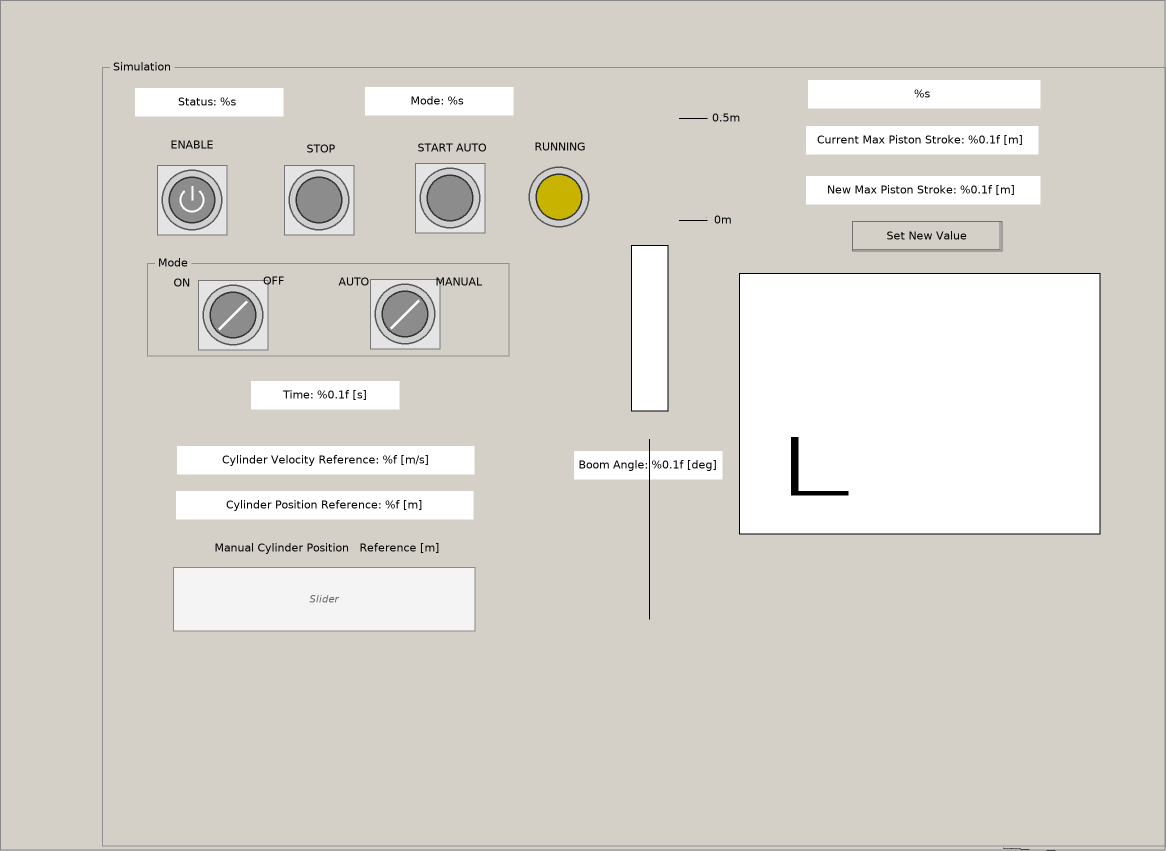
VISUALIZATION CraneHMI  // 1166x851
    Rectangle (566,310 166x37), angle 270
    GroupBox (102,59 1064x787), "Simulation"
        GroupBox (45,196 362x101), "Mode"
        Rectangle (637,214 361x261)
        PowerSwitch (55,106 70x70), variable: HMI.bPowerOn, behaviour: TOGGLE, style: Switch-PowerSwitch-Gray
        PushSwitch (313,104 70x70), variable: HMI.bStart, behaviour: TAP, style: Switch-PushSwitch-Gray
        Lamp1 (422,103 70x70), variable: HMI.bRunning, style: Lamp-Lamp1-Yellow
        Textfield (74,386 299x30), "Cylinder Velocity Reference: %f [m/s]", text variable: HMI.fCylinderVelocityReference
            OnMouseClick: write the text variable via Default
        Label (15,71 150x30), "ENABLE"
        Label (275,74 150x30), "START AUTO"
        Label (383,73 150x30), "RUNNING"
        Textfield (148,321 150x30), "Time: %0.1f [s]", text variable: HMI.fSimulationTime
        Label (90,474 270x30), "Manual Cylinder Position Reference [m]"
        Textfield (73,431 299x30), "Cylinder Position Reference: %f [m]", text variable: HMI.fCylinderPosition
        Line (577,161) (605,161)
        Label (607,146 28x30), "0m"
        Textfield (703,66 234x30), "Current Max Piston Stroke: %0.1f [m]", text variable: Parameters.stParam.stPistonRange.fPistonPosMax
        Textfield (703,116 236x30), "New Max Piston Stroke: %0.1f [m]", text variable: HMI.fMaxPistonPosition
            OnMouseDown: write the text variable via Default, min 0, max 1
        Button (750,162 150x30), "Set New Value"
            tap CraneSimulation.bPistonMaxNewValue
        Line (577,59) (605,59)
        Textfield (32,28 150x30), "Status: %s", text variable: HMI.eStatus
        Textfield (262,27 150x30), "Mode: %s", text variable: HMI.eMode
        Textfield (705,20 234x30), "%s", text variable: HMI.sPistonEndStopMessages
        Textfield (471,391 150x30), "Boom Angle: %0.1f [deg]", text variable: HMI.fBoomAngleDeg
        Slider (71,508 302x64), variable: HMI.fManualCylinderPositionReference, scale 0..0.5
        Rectangle (689,378 7x58)
        Rectangle (690,432 56x4)
        RotarySwitch (96,221 70x70), variable: HMI.bOn, behaviour: TOGGLE, style: Switch-RotarySwitch-Gray
        RotarySwitch (268,220 70x70), variable: HMI.bAuto, behaviour: TOGGLE, style: Switch-RotarySwitch-Gray
        Label (282,208 150x30), "MANUAL"
        Label (177,208 150x30), "AUTO"
        Label (97,207 150x30), "OFF"
        PushSwitch (182,106 70x70), variable: HMI.bStop, behaviour: TAP, style: Switch-PushSwitch-Gray
        Label (144,75 150x30), "STOP"
    Line (649,439) (649,619)
        p1126004900: HMI.stPistonAnimation.pt1_y
        p3528305787: HMI.stPistonAnimation.pt0_x
        p2773130477: HMI.stPistonAnimation.pt0_y
        p874137650: HMI.stPistonAnimation.pt1_x
    Line (706,217) (706,217)
    Label (712,103 28x30), "0.5m"
    Line (721,115) (721,115)
    Line (1055,851) (1003,848)
        p1126004900: HMI.stBoomAnimation.pt1_y
        p3528305787: HMI.stBoomAnimation.pt0_x
        p2773130477: HMI.stBoomAnimation.pt0_y
        p874137650: -HMI.stBoomAnimation.pt1_x
    Label (107,268 150x30), "ON"
END_VISUALIZATION

(* stored: Version 1.1.0.1, ProductVersion 3.1.4024.10
   Visu CraneHMI: Id {4bdd8ed7-7379-4dd1-955f-a8a1c50d5ff4} *)
